// TIA Portal V17 export
// export: Created 2025-08-05T09:36:00.7805408Z, ExportSetting WithDefaults, DisplayName Totally Integrated Automation Portal, DisplayVersion V17, DisplayName TIA Portal Openness, DisplayVersion V17, DisplayName TIA Portal Version Control Interface, DisplayVersion V17, DisplayName SINAMICS Startdrive Advanced, DisplayVersion V17, DisplayName SINAMICS Startdrive G130, G150, S120, S150, SINAMICS MV, S210, DisplayVersion V17, DisplayName SINAMICS Startdrive G110M, G120, G120C, G120D, G120P, G115D, DisplayVersion V17, DisplayName STEP 7 Professional, DisplayVersion V17, DisplayName STEP 7 Safety, DisplayVersion V17, DisplayName WinCC Advanced, DisplayVersion V17
TYPE "typeTeststoppSBTData"
// V 01.00
// stored: IsFailsafeCompliant false
   STRUCT
      BrakeTestRequest { S7_SetPoint := 'True'} : Bool := false;   // Bremsentest Anforderung / Brake test request
      BrakeTestRequestWithPreconditions : Bool;   // Bremsentest Anforderung mit Vorbedingungen / Brake test request with preconditions
      BrakeTestPreconditionsNOK : Bool;   // Bremsentest Vorbedingungen NOK / Brake test preconditions NOK
      BrakeTestImmediately { S7_SetPoint := 'True'} : Bool := false;   // Sofortausführung Bremsentest / Immediate execution brake test
      BrakeTestActive : Bool;   // Bremsentest ist zur Zeit aktiv / Brake test is currently active
      SafeGuardBlocked { S7_SetPoint := 'True'} : Bool := false;   // Öffnen/Entriegeln der Schutzteinrichtung ist geblockt / Opening/unlocking the safeguard is blocked
   END_STRUCT;
END_TYPE
